DATA_BLOCK "ST10_MaterialGate4_DB"
{ S7_Optimized_Access := 'FALSE' }
VERSION : 0.1
NON_RETAIN
// ATTRIBUTES
// AUTO_NUMBER = False
// BLOCK_NUMBER = 1154
// END_ATTRIBUTES
"SafetyGate"

BEGIN

END_DATA_BLOCK

